FUNCTION_BLOCK FB_masterConnectionCheck
VAR
	// current state 
	m_isConnected :BOOL :=FALSE;
	
	// last heart beat
	m_lastHeartBeat :INT:=0 ;
	
	// current conneciton cycles
	m_curConnectionCycles :INT:=0;
	
	// current disconneciton cycles
	m_curDisconnectionCycles :INT:=0;
	
	// conneciton cycles thresshold
	m_connectionCyclesThres :INT:=5;
	
END_VAR

METHOD PUBLIC check : BOOL
VAR_INPUT
	i_heartBeat :INT;
END_VAR
// current is disconnected
IF NOT(m_isConnected) THEN
	m_curDisconnectionCycles:=0;
	
	IF  i_heartBeat <> m_lastHeartBeat THEN
		m_curConnectionCycles :=  m_curConnectionCycles +1;
	ELSE
		m_curConnectionCycles :=0;
	END_IF
	
	IF  m_curConnectionCycles >= m_connectionCyclesThres THEN
		m_isConnected := TRUE;
	END_IF

// current is connected
ELSE
	m_curConnectionCycles :=0;
	
	IF  i_heartBeat = m_lastHeartBeat THEN
		m_curDisconnectionCycles := m_curDisconnectionCycles +1;
	ELSE
		m_curDisconnectionCycles :=0;
	END_IF
	
	IF m_curDisconnectionCycles>= m_connectionCyclesThres THEN
		m_isConnected:=FALSE;
	END_IF

END_IF

m_lastHeartBeat:= i_heartBeat;
check:=m_isConnected;
END_METHOD

END_FUNCTION_BLOCK

(* stored: Version 1.1.0.1, ProductVersion 3.1.4024.11
   POU FB_masterConnectionCheck: Id {e5f1fdfc-6a14-4f4a-8041-8bb9448142d8}, SpecialFunc None
   Method check: Id {637c8591-2caa-40e8-9a5f-7460ac421fa8} *)
